Universal Robots PolyScope program: random_move_in_box_xmlrpc.urp

Program random_move_in_box_xmlrpc (installation=default directory=/programs/Stable createdIn=5.9.1.1031110 lastSavedIn=5.10.0.106288 robotSerialNumber=20185500256)
Calibrated DH parameters: a=[0.000163, -0.146131, -0.38577, 0.000126, -0.000021, 0]; d=[0.161954, 188.306531, -157.478086, -30.695088, 0.099716, 0.099628]; alpha=[1.569701, -0.00212, 0.002263, 1.570438, -1.570123, 0]; deltaTheta=[0, -1.219859, 7.681919, -0.178877, -0.000001, 0]
InitVariablesNode
BeforeStart
  Call URCancelManualMove
  MoveJ speed 60 deg/s, acceleration 80 deg/s^2 (useActiveTCP=true positionType=JointAngles) feature=Base
    Waypoint HomeWP: TCP in base x=132.769 y=-491.632 z=236.295 mm, rx=0.0018 ry=-3.1384 rz=0.0008 rad; joints [90.004, -89.995, 90.002, -89.997, -90.004, 0.023] deg; TCP offset x=0 y=0 z=250.5 mm, rx=0 ry=0 rz=0 rad
  Call InitGripper
Robot Program (runOnlyOnce=false)
  'MoveJ in script line as it enables seeding the numeric inverse kinematics solver'
  Script: movej(get_inverse_kin(cam_bin1, HomeWP_q))
  URCap XML-RPC Call (DTI UR Helper, Danish Technological Institute) dataModel(xmlrpc_function=get_grasp_pose, xmlrpc_handle=train); state(isChildrenLocked=true)
    result := train.get_grasp_pose()
  x := result[0]
  y := result[1]
  rz := result[2]
  d := result[3]
  Call SetGripperWidth
  Call MoveToApproach
  Call MoveAndGrasp
  Call MoveToSafety
  If egiGripped()
    'MoveJ in script line as it enables seeding the numeric inverse kinematics solver'
    Script: movej(get_inverse_kin(cam_bin2, HomeWP_q))
    URCap EGI Grip (SCHUNK Gripper EGI for UR, SCHUNK GmbH & Co.) dataModel(use_work_piece=true, async_exe=true, grip_type=3)
  Else 
    d := 1
    Call SetGripperWidth
  SuppressedNode
    Call MoveToSafety
SubProgram  [hidden by the author, left out]
SubProgram  [hidden by the author, left out]
SubProgram  [hidden by the author, left out]
SubProgram  [hidden by the author, left out]
SubProgram  [hidden by the author, left out]
SubProgram  [hidden by the author, left out]
SubProgram URCancelManualMove [hidden by the author, left out]
SubProgram InitGripper [hidden by the author, left out]
SubProgram SetGripperWidth [hidden by the author, left out]
SubProgram MoveToApproach [hidden by the author, left out]
SubProgram MoveAndGrasp [hidden by the author, left out]
SubProgram MoveToSafety [hidden by the author, left out]
